FUNCTION_BLOCK PLCopenNullRemote IMPLEMENTS IPLCopenCall

// Copyright (c) 2024 Loupe (https://loupe.team), provided under the MIT License.

METHOD Aborted : BOOL
// Copyright (c) 2024 Loupe (https://loupe.team), provided under the MIT License.
END_METHOD

METHOD Errored : BOOL
VAR_INPUT
    ID : INT;
END_VAR
// Copyright (c) 2024 Loupe (https://loupe.team), provided under the MIT License.
END_METHOD

METHOD Finished : BOOL
// Copyright (c) 2024 Loupe (https://loupe.team), provided under the MIT License.
END_METHOD

{warning 'add method implementation '}
METHOD Start : BOOL
VAR_INPUT
    Command : IPLCopenCommand;
END_VAR
// Copyright (c) 2024 Loupe (https://loupe.team), provided under the MIT License.

//TODO
END_METHOD

END_FUNCTION_BLOCK

(* stored: Version 1.1.0.1
   POU PLCopenNullRemote: Id {73061230-7a8e-410b-ae26-c14eb801f0aa}, SpecialFunc None
   Method Aborted: Id {d3377050-9f4c-49f6-a051-4bcdc44d847d}
   Method Errored: Id {97c3ac24-72bd-4b21-93c4-11f805822d38}
   Method Finished: Id {6fdf66c9-5086-43d9-b213-c69b23218cc4}
   Method Start: Id {42d0f9af-461f-4d36-bb4c-e7ed19b6748a} *)
